FUNCTION_BLOCK FB_Blink
VAR_INPUT
	i_sName	: STRING;
	i_bEnable: BOOL;
	i_tTime: TIME := T#1S;
END_VAR
VAR_OUTPUT
	o_bOut: BOOL;
END_VAR
VAR
	T1_TON: TON;
	T2_TOF: TOF;
END_VAR

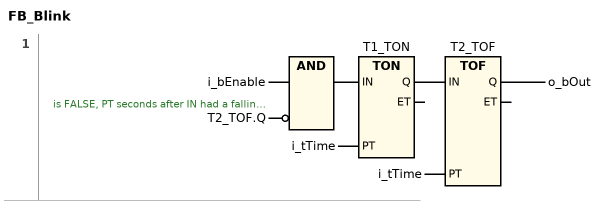
// NETWORK 1
//   T2_TOF.Q: is FALSE, PT seconds after IN had a falling edge
T1_TON(IN := i_bEnable AND NOT T2_TOF.Q, PT := i_tTime); // TON
T2_TOF(IN := T1_TON.Q, PT := i_tTime); // TOF
o_bOut := T2_TOF.Q;

END_FUNCTION_BLOCK

(* stored: Version 1.1.0.1, ProductVersion 3.1.4022.6
   POU FB_Blink: Id {b13e67f6-e1fd-4bfe-85ae-fabaf3144d97}, SpecialFunc None *)
